// TIA Portal V21 export
FUNCTION "CipEvents" : Void   // FC2, LAD
{ S7_Optimized_Access := 'TRUE' }
// stored: SetENOAutomatically false
   VAR_TEMP   // added for the SCL form of the ladder/FBD networks
      _w1 : Bool;
      _w2 : Bool;
      _w3 : Bool;
      _w4 : Bool;
      _w5 : Bool;
      _w6 : Bool;
      _w7 : Bool;
      _w8 : Bool;
      _w9 : Bool;
      _w10 : Bool;
      _w11 : Bool;
      _w12 : Bool;
      _w13 : Bool;
      _w14 : Bool;
      _w15 : Bool;
      _w16 : Bool;
      _w17 : Bool;
      _w18 : Bool;
      _w19 : Bool;
      _w20 : Bool;
      _w21 : Bool;
      _w22 : Bool;
      _w23 : Bool;
      _w24 : Bool;
      _w25 : Bool;
      _w26 : Bool;
      _w27 : Bool;
      _w28 : Bool;
      _w29 : Bool;
      _w30 : Bool;
      _w31 : Bool;
      _w32 : Bool;
      _w33 : Bool;
      _w34 : Bool;
      _w35 : Bool;
      _w36 : Bool;
      _w37 : Bool;
      _w38 : Bool;
      _w39 : Bool;
      _w40 : Bool;
   END_VAR
BEGIN

REGION Network 1: ****************D500****************
END_REGION

REGION Network 2: Events And Line Print
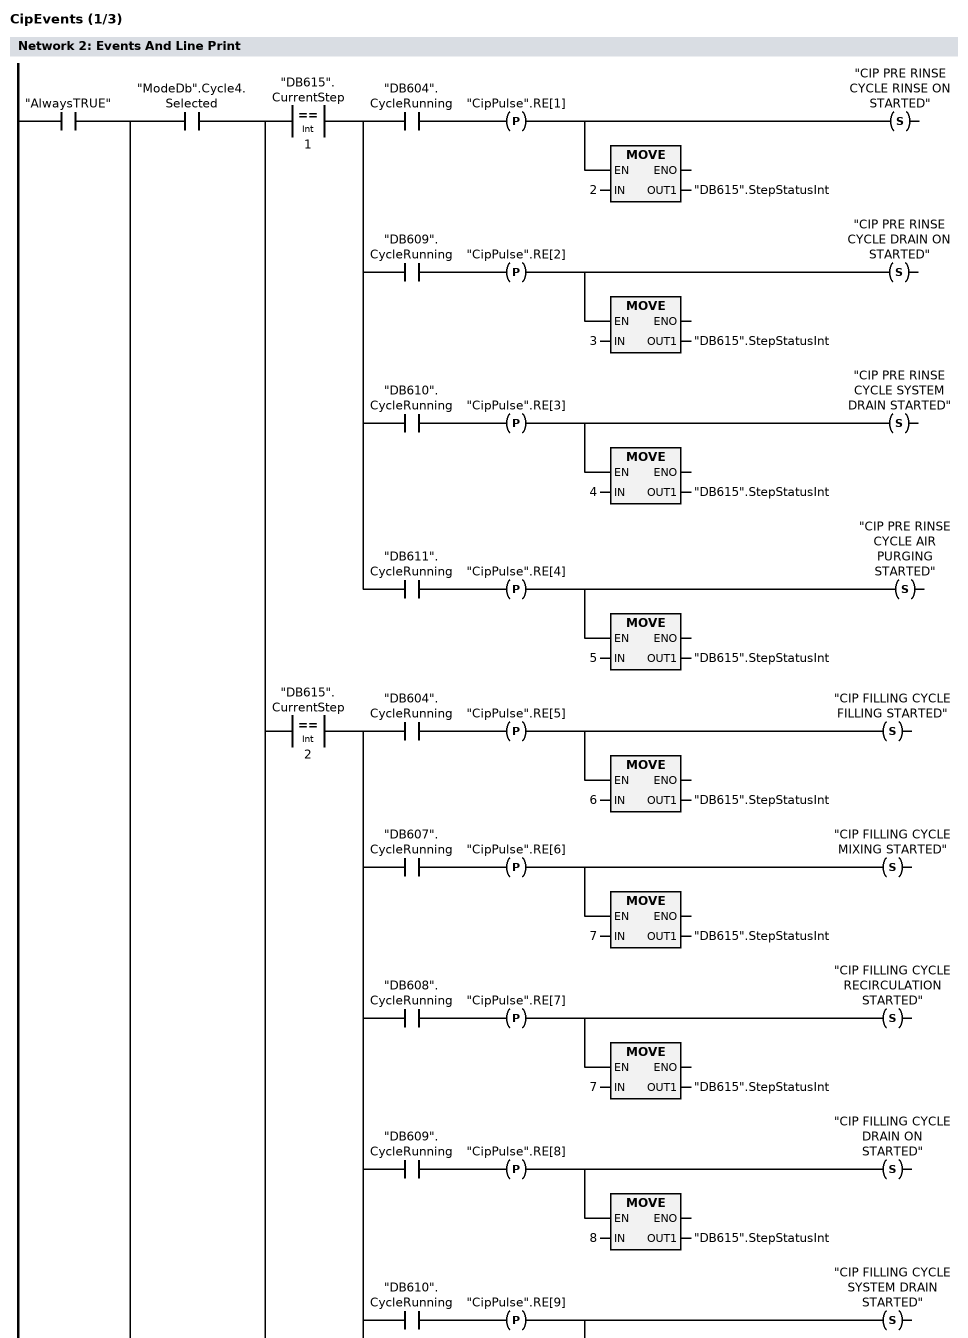
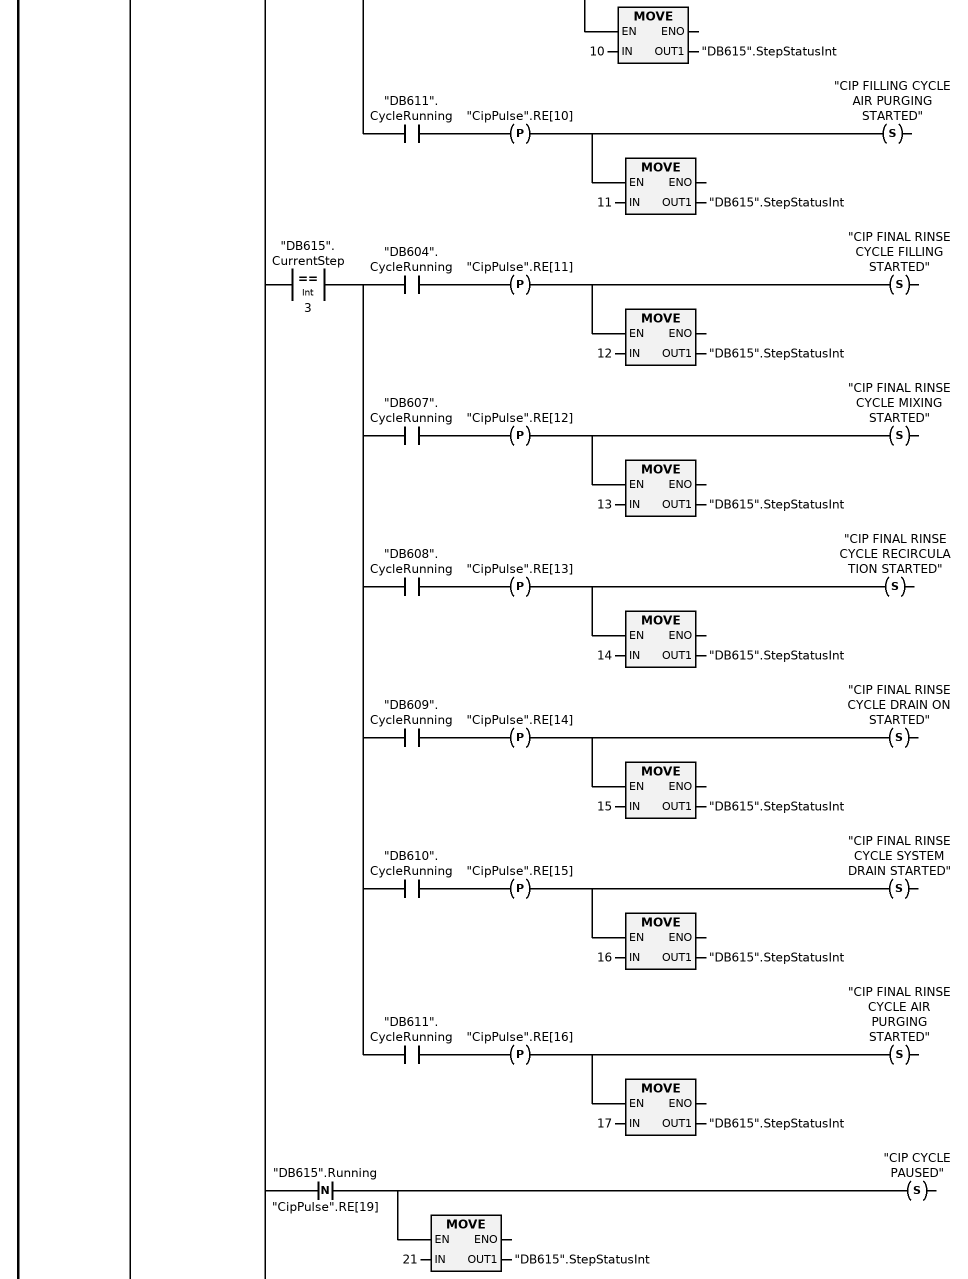
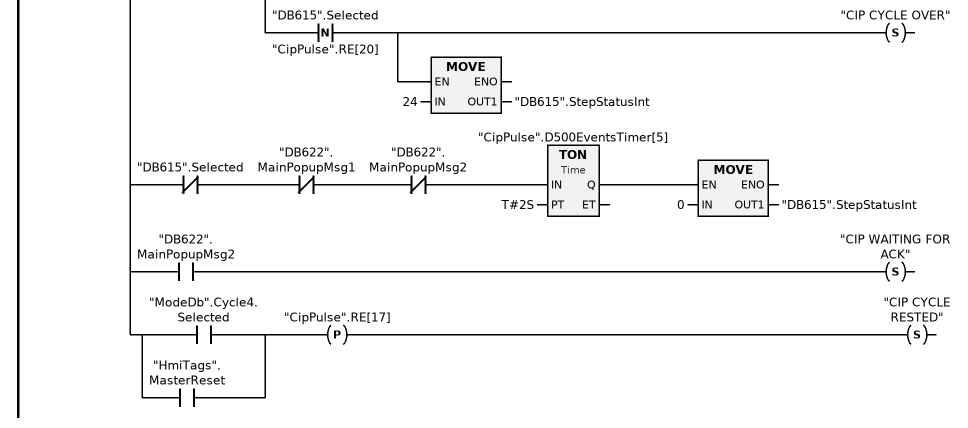
   RUNG wire#powerrail
      Contact( "AlwaysTRUE" )
      wire#w1
      Contact( "ModeDb".Cycle4.Selected )
      wire#w2
      { S7_Templates := "SrcType := Int" } EQ_Contact(in1 := "DB615".CurrentStep, in2 := 1)
      wire#w3
      Contact( "DB604".CycleRunning )
      P_Trig( "CipPulse".RE[1] )
      wire#w4
      S_Coil( "CIP PRE RINSE CYCLE RINSE ON STARTED" )
   END_RUNG
   RUNG wire#w4
      Move(in := 2, out1 => "DB615".StepStatusInt)
   END_RUNG
   RUNG wire#w3
      Contact( "DB609".CycleRunning )
      P_Trig( "CipPulse".RE[2] )
      wire#w5
      S_Coil( "CIP PRE RINSE CYCLE DRAIN ON STARTED" )
   END_RUNG
   RUNG wire#w5
      Move(in := 3, out1 => "DB615".StepStatusInt)
   END_RUNG
   RUNG wire#w3
      Contact( "DB610".CycleRunning )
      P_Trig( "CipPulse".RE[3] )
      wire#w6
      S_Coil( "CIP PRE RINSE CYCLE SYSTEM DRAIN STARTED" )
   END_RUNG
   RUNG wire#w6
      Move(in := 4, out1 => "DB615".StepStatusInt)
   END_RUNG
   RUNG wire#w3
      Contact( "DB611".CycleRunning )
      P_Trig( "CipPulse".RE[4] )
      wire#w7
      S_Coil( "CIP PRE RINSE CYCLE AIR PURGING STARTED" )
   END_RUNG
   RUNG wire#w7
      Move(in := 5, out1 => "DB615".StepStatusInt)
   END_RUNG
   RUNG wire#w2
      { S7_Templates := "SrcType := Int" } EQ_Contact(in1 := "DB615".CurrentStep, in2 := 2)
      wire#w8
      Contact( "DB604".CycleRunning )
      P_Trig( "CipPulse".RE[5] )
      wire#w9
      S_Coil( "CIP FILLING CYCLE FILLING STARTED" )
   END_RUNG
   RUNG wire#w9
      Move(in := 6, out1 => "DB615".StepStatusInt)
   END_RUNG
   RUNG wire#w8
      Contact( "DB607".CycleRunning )
      P_Trig( "CipPulse".RE[6] )
      wire#w10
      S_Coil( "CIP FILLING CYCLE MIXING STARTED" )
   END_RUNG
   RUNG wire#w10
      Move(in := 7, out1 => "DB615".StepStatusInt)
   END_RUNG
   RUNG wire#w8
      Contact( "DB608".CycleRunning )
      P_Trig( "CipPulse".RE[7] )
      wire#w11
      S_Coil( "CIP FILLING CYCLE RECIRCULATION STARTED" )
   END_RUNG
   RUNG wire#w11
      Move(in := 7, out1 => "DB615".StepStatusInt)
   END_RUNG
   RUNG wire#w8
      Contact( "DB609".CycleRunning )
      P_Trig( "CipPulse".RE[8] )
      wire#w12
      S_Coil( "CIP FILLING CYCLE DRAIN ON STARTED" )
   END_RUNG
   RUNG wire#w12
      Move(in := 8, out1 => "DB615".StepStatusInt)
   END_RUNG
   RUNG wire#w8
      Contact( "DB610".CycleRunning )
      P_Trig( "CipPulse".RE[9] )
      wire#w13
      S_Coil( "CIP FILLING CYCLE SYSTEM DRAIN STARTED" )
   END_RUNG
   RUNG wire#w13
      Move(in := 10, out1 => "DB615".StepStatusInt)
   END_RUNG
   RUNG wire#w8
      Contact( "DB611".CycleRunning )
      P_Trig( "CipPulse".RE[10] )
      wire#w14
      S_Coil( "CIP FILLING CYCLE AIR PURGING STARTED" )
   END_RUNG
   RUNG wire#w14
      Move(in := 11, out1 => "DB615".StepStatusInt)
   END_RUNG
   RUNG wire#w2
      { S7_Templates := "SrcType := Int" } EQ_Contact(in1 := "DB615".CurrentStep, in2 := 3)
      wire#w15
      Contact( "DB604".CycleRunning )
      P_Trig( "CipPulse".RE[11] )
      wire#w16
      S_Coil( "CIP FINAL RINSE CYCLE FILLING STARTED" )
   END_RUNG
   RUNG wire#w16
      Move(in := 12, out1 => "DB615".StepStatusInt)
   END_RUNG
   RUNG wire#w15
      Contact( "DB607".CycleRunning )
      P_Trig( "CipPulse".RE[12] )
      wire#w17
      S_Coil( "CIP FINAL RINSE CYCLE MIXING STARTED" )
   END_RUNG
   RUNG wire#w17
      Move(in := 13, out1 => "DB615".StepStatusInt)
   END_RUNG
   RUNG wire#w15
      Contact( "DB608".CycleRunning )
      P_Trig( "CipPulse".RE[13] )
      wire#w18
      S_Coil( "CIP FINAL RINSE CYCLE RECIRCULATION STARTED" )
   END_RUNG
   RUNG wire#w18
      Move(in := 14, out1 => "DB615".StepStatusInt)
   END_RUNG
   RUNG wire#w15
      Contact( "DB609".CycleRunning )
      P_Trig( "CipPulse".RE[14] )
      wire#w19
      S_Coil( "CIP FINAL RINSE CYCLE DRAIN ON STARTED" )
   END_RUNG
   RUNG wire#w19
      Move(in := 15, out1 => "DB615".StepStatusInt)
   END_RUNG
   RUNG wire#w15
      Contact( "DB610".CycleRunning )
      P_Trig( "CipPulse".RE[15] )
      wire#w20
      S_Coil( "CIP FINAL RINSE CYCLE SYSTEM DRAIN STARTED" )
   END_RUNG
   RUNG wire#w20
      Move(in := 16, out1 => "DB615".StepStatusInt)
   END_RUNG
   RUNG wire#w15
      Contact( "DB611".CycleRunning )
      P_Trig( "CipPulse".RE[16] )
      wire#w21
      S_Coil( "CIP FINAL RINSE CYCLE AIR PURGING STARTED" )
   END_RUNG
   RUNG wire#w21
      Move(in := 17, out1 => "DB615".StepStatusInt)
   END_RUNG
   RUNG wire#w2
      N_Contact(operand := "DB615".Running, bit := "CipPulse".RE[19])
      wire#w22
      S_Coil( "CIP CYCLE PAUSED" )
   END_RUNG
   RUNG wire#w22
      Move(in := 21, out1 => "DB615".StepStatusInt)
   END_RUNG
   RUNG wire#w2
      N_Contact(operand := "DB615".Selected, bit := "CipPulse".RE[20])
      wire#w23
      S_Coil( "CIP CYCLE OVER" )
   END_RUNG
   RUNG wire#w23
      Move(in := 24, out1 => "DB615".StepStatusInt)
   END_RUNG
   RUNG wire#w1
      I_Contact( "DB615".Selected )
      I_Contact( "DB622".MainPopupMsg1 )
      I_Contact( "DB622".MainPopupMsg2 )
      { S7_Templates := "time_type := Time" } "CipPulse".D500EventsTimer[5].TON(pt := T#2S, et =>)
      Move(in := 0, out1 => "DB615".StepStatusInt)
   END_RUNG
   RUNG wire#w1
      Contact( "DB622".MainPopupMsg2 )
      S_Coil( "CIP WAITING FOR ACK" )
   END_RUNG
   RUNG wire#w1
      Contact( "ModeDb".Cycle4.Selected )
      wire#w24
      P_Trig( "CipPulse".RE[17] )
      S_Coil( "CIP CYCLE RESTED" )
   END_RUNG
   RUNG wire#w1
      Contact( "HmiTags".MasterReset )
   END_RUNG wire#w24
   // the same network as SCL:
   #_w1 := "AlwaysTRUE" AND "ModeDb".Cycle4.Selected;
   #_w2 := #_w1 AND ("DB615".CurrentStep = 1);
   #_w3 := #_w2 AND "DB604".CycleRunning;
   #_w4 := #_w3 AND NOT "CipPulse".RE[1];   // rising edge
   "CipPulse".RE[1] := #_w3;
   IF #_w4 THEN
       "CIP PRE RINSE CYCLE RINSE ON STARTED" := TRUE;
       "DB615".StepStatusInt := 2;
   END_IF;
   #_w5 := #_w2 AND "DB609".CycleRunning;
   #_w6 := #_w5 AND NOT "CipPulse".RE[2];   // rising edge
   "CipPulse".RE[2] := #_w5;
   IF #_w6 THEN
       "CIP PRE RINSE CYCLE DRAIN ON STARTED" := TRUE;
       "DB615".StepStatusInt := 3;
   END_IF;
   #_w7 := #_w2 AND "DB610".CycleRunning;
   #_w8 := #_w7 AND NOT "CipPulse".RE[3];   // rising edge
   "CipPulse".RE[3] := #_w7;
   IF #_w8 THEN
       "CIP PRE RINSE CYCLE SYSTEM DRAIN STARTED" := TRUE;
       "DB615".StepStatusInt := 4;
   END_IF;
   #_w9 := #_w2 AND "DB611".CycleRunning;
   #_w10 := #_w9 AND NOT "CipPulse".RE[4];   // rising edge
   "CipPulse".RE[4] := #_w9;
   IF #_w10 THEN
       "CIP PRE RINSE CYCLE AIR PURGING STARTED" := TRUE;
       "DB615".StepStatusInt := 5;
   END_IF;
   #_w11 := #_w1 AND ("DB615".CurrentStep = 2);
   #_w12 := #_w11 AND "DB604".CycleRunning;
   #_w13 := #_w12 AND NOT "CipPulse".RE[5];   // rising edge
   "CipPulse".RE[5] := #_w12;
   IF #_w13 THEN
       "CIP FILLING CYCLE FILLING STARTED" := TRUE;
       "DB615".StepStatusInt := 6;
   END_IF;
   #_w14 := #_w11 AND "DB607".CycleRunning;
   #_w15 := #_w14 AND NOT "CipPulse".RE[6];   // rising edge
   "CipPulse".RE[6] := #_w14;
   IF #_w15 THEN
       "CIP FILLING CYCLE MIXING STARTED" := TRUE;
       "DB615".StepStatusInt := 7;
   END_IF;
   #_w16 := #_w11 AND "DB608".CycleRunning;
   #_w17 := #_w16 AND NOT "CipPulse".RE[7];   // rising edge
   "CipPulse".RE[7] := #_w16;
   IF #_w17 THEN
       "CIP FILLING CYCLE RECIRCULATION STARTED" := TRUE;
       "DB615".StepStatusInt := 7;
   END_IF;
   #_w18 := #_w11 AND "DB609".CycleRunning;
   #_w19 := #_w18 AND NOT "CipPulse".RE[8];   // rising edge
   "CipPulse".RE[8] := #_w18;
   IF #_w19 THEN
       "CIP FILLING CYCLE DRAIN ON STARTED" := TRUE;
       "DB615".StepStatusInt := 8;
   END_IF;
   #_w20 := #_w11 AND "DB610".CycleRunning;
   #_w21 := #_w20 AND NOT "CipPulse".RE[9];   // rising edge
   "CipPulse".RE[9] := #_w20;
   IF #_w21 THEN
       "CIP FILLING CYCLE SYSTEM DRAIN STARTED" := TRUE;
       "DB615".StepStatusInt := 10;
   END_IF;
   #_w22 := #_w11 AND "DB611".CycleRunning;
   #_w23 := #_w22 AND NOT "CipPulse".RE[10];   // rising edge
   "CipPulse".RE[10] := #_w22;
   IF #_w23 THEN
       "CIP FILLING CYCLE AIR PURGING STARTED" := TRUE;
       "DB615".StepStatusInt := 11;
   END_IF;
   #_w24 := #_w1 AND ("DB615".CurrentStep = 3);
   #_w25 := #_w24 AND "DB604".CycleRunning;
   #_w26 := #_w25 AND NOT "CipPulse".RE[11];   // rising edge
   "CipPulse".RE[11] := #_w25;
   IF #_w26 THEN
       "CIP FINAL RINSE CYCLE FILLING STARTED" := TRUE;
       "DB615".StepStatusInt := 12;
   END_IF;
   #_w27 := #_w24 AND "DB607".CycleRunning;
   #_w28 := #_w27 AND NOT "CipPulse".RE[12];   // rising edge
   "CipPulse".RE[12] := #_w27;
   IF #_w28 THEN
       "CIP FINAL RINSE CYCLE MIXING STARTED" := TRUE;
       "DB615".StepStatusInt := 13;
   END_IF;
   #_w29 := #_w24 AND "DB608".CycleRunning;
   #_w30 := #_w29 AND NOT "CipPulse".RE[13];   // rising edge
   "CipPulse".RE[13] := #_w29;
   IF #_w30 THEN
       "CIP FINAL RINSE CYCLE RECIRCULATION STARTED" := TRUE;
       "DB615".StepStatusInt := 14;
   END_IF;
   #_w31 := #_w24 AND "DB609".CycleRunning;
   #_w32 := #_w31 AND NOT "CipPulse".RE[14];   // rising edge
   "CipPulse".RE[14] := #_w31;
   IF #_w32 THEN
       "CIP FINAL RINSE CYCLE DRAIN ON STARTED" := TRUE;
       "DB615".StepStatusInt := 15;
   END_IF;
   #_w33 := #_w24 AND "DB610".CycleRunning;
   #_w34 := #_w33 AND NOT "CipPulse".RE[15];   // rising edge
   "CipPulse".RE[15] := #_w33;
   IF #_w34 THEN
       "CIP FINAL RINSE CYCLE SYSTEM DRAIN STARTED" := TRUE;
       "DB615".StepStatusInt := 16;
   END_IF;
   #_w35 := #_w24 AND "DB611".CycleRunning;
   #_w36 := #_w35 AND NOT "CipPulse".RE[16];   // rising edge
   "CipPulse".RE[16] := #_w35;
   IF #_w36 THEN
       "CIP FINAL RINSE CYCLE AIR PURGING STARTED" := TRUE;
       "DB615".StepStatusInt := 17;
   END_IF;
   #_w37 := #_w1 AND NOT "DB615".Running AND "CipPulse".RE[19];   // falling edge of "DB615".Running
   "CipPulse".RE[19] := "DB615".Running;
   IF #_w37 THEN
       "CIP CYCLE PAUSED" := TRUE;
       "DB615".StepStatusInt := 21;
   END_IF;
   #_w38 := #_w1 AND NOT "DB615".Selected AND "CipPulse".RE[20];   // falling edge of "DB615".Selected
   "CipPulse".RE[20] := "DB615".Selected;
   IF #_w38 THEN
       "CIP CYCLE OVER" := TRUE;
       "DB615".StepStatusInt := 24;
   END_IF;
   "CipPulse".D500EventsTimer[5].TON(IN := "AlwaysTRUE" AND NOT "DB615".Selected AND NOT "DB622".MainPopupMsg1 AND NOT "DB622".MainPopupMsg2,
                           PT := T#2S);
   IF "CipPulse".D500EventsTimer[5].Q THEN "DB615".StepStatusInt := 0; END_IF;
   IF "AlwaysTRUE" AND "DB622".MainPopupMsg2 THEN "CIP WAITING FOR ACK" := TRUE; END_IF;
   #_w39 := "AlwaysTRUE" AND ("ModeDb".Cycle4.Selected OR "HmiTags".MasterReset);
   #_w40 := #_w39 AND NOT "CipPulse".RE[17];   // rising edge
   "CipPulse".RE[17] := #_w39;
   IF #_w40 THEN "CIP CYCLE RESTED" := TRUE; END_IF;
END_REGION

REGION Network 3: PRE RINSE
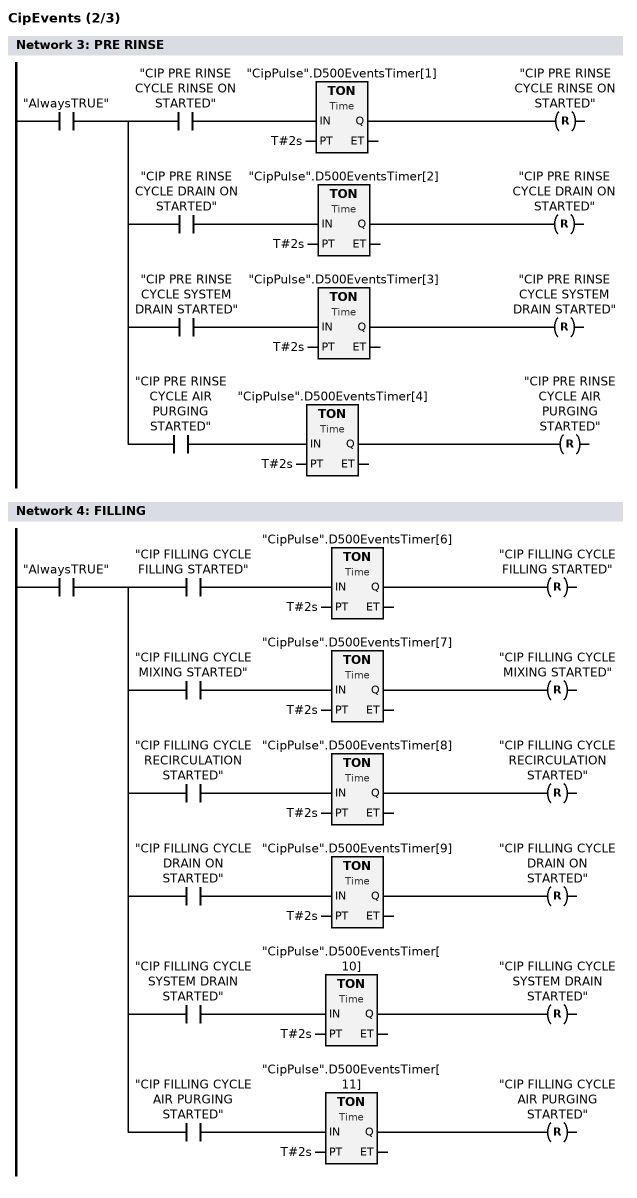
   RUNG wire#powerrail
      Contact( "AlwaysTRUE" )
      wire#w1
      Contact( "CIP PRE RINSE CYCLE RINSE ON STARTED" )
      { S7_Templates := "time_type := Time" } "CipPulse".D500EventsTimer[1].TON(pt := T#2s, et =>)
      R_Coil( "CIP PRE RINSE CYCLE RINSE ON STARTED" )
   END_RUNG
   RUNG wire#w1
      Contact( "CIP PRE RINSE CYCLE DRAIN ON STARTED" )
      { S7_Templates := "time_type := Time" } "CipPulse".D500EventsTimer[2].TON(pt := T#2s, et =>)
      R_Coil( "CIP PRE RINSE CYCLE DRAIN ON STARTED" )
   END_RUNG
   RUNG wire#w1
      Contact( "CIP PRE RINSE CYCLE SYSTEM DRAIN STARTED" )
      { S7_Templates := "time_type := Time" } "CipPulse".D500EventsTimer[3].TON(pt := T#2s, et =>)
      R_Coil( "CIP PRE RINSE CYCLE SYSTEM DRAIN STARTED" )
   END_RUNG
   RUNG wire#w1
      Contact( "CIP PRE RINSE CYCLE AIR PURGING STARTED" )
      { S7_Templates := "time_type := Time" } "CipPulse".D500EventsTimer[4].TON(pt := T#2s, et =>)
      R_Coil( "CIP PRE RINSE CYCLE AIR PURGING STARTED" )
   END_RUNG
   // the same network as SCL:
   "CipPulse".D500EventsTimer[1].TON(IN := "AlwaysTRUE" AND "CIP PRE RINSE CYCLE RINSE ON STARTED", PT := T#2s);
   IF "CipPulse".D500EventsTimer[1].Q THEN "CIP PRE RINSE CYCLE RINSE ON STARTED" := FALSE; END_IF;
   "CipPulse".D500EventsTimer[2].TON(IN := "AlwaysTRUE" AND "CIP PRE RINSE CYCLE DRAIN ON STARTED", PT := T#2s);
   IF "CipPulse".D500EventsTimer[2].Q THEN "CIP PRE RINSE CYCLE DRAIN ON STARTED" := FALSE; END_IF;
   "CipPulse".D500EventsTimer[3].TON(IN := "AlwaysTRUE" AND "CIP PRE RINSE CYCLE SYSTEM DRAIN STARTED",
                           PT := T#2s);
   IF "CipPulse".D500EventsTimer[3].Q THEN "CIP PRE RINSE CYCLE SYSTEM DRAIN STARTED" := FALSE; END_IF;
   "CipPulse".D500EventsTimer[4].TON(IN := "AlwaysTRUE" AND "CIP PRE RINSE CYCLE AIR PURGING STARTED",
                           PT := T#2s);
   IF "CipPulse".D500EventsTimer[4].Q THEN "CIP PRE RINSE CYCLE AIR PURGING STARTED" := FALSE; END_IF;
END_REGION

REGION Network 4: FILLING
   RUNG wire#powerrail
      Contact( "AlwaysTRUE" )
      wire#w1
      Contact( "CIP FILLING CYCLE FILLING STARTED" )
      { S7_Templates := "time_type := Time" } "CipPulse".D500EventsTimer[6].TON(pt := T#2s, et =>)
      R_Coil( "CIP FILLING CYCLE FILLING STARTED" )
   END_RUNG
   RUNG wire#w1
      Contact( "CIP FILLING CYCLE MIXING STARTED" )
      { S7_Templates := "time_type := Time" } "CipPulse".D500EventsTimer[7].TON(pt := T#2s, et =>)
      R_Coil( "CIP FILLING CYCLE MIXING STARTED" )
   END_RUNG
   RUNG wire#w1
      Contact( "CIP FILLING CYCLE RECIRCULATION STARTED" )
      { S7_Templates := "time_type := Time" } "CipPulse".D500EventsTimer[8].TON(pt := T#2s, et =>)
      R_Coil( "CIP FILLING CYCLE RECIRCULATION STARTED" )
   END_RUNG
   RUNG wire#w1
      Contact( "CIP FILLING CYCLE DRAIN ON STARTED" )
      { S7_Templates := "time_type := Time" } "CipPulse".D500EventsTimer[9].TON(pt := T#2s, et =>)
      R_Coil( "CIP FILLING CYCLE DRAIN ON STARTED" )
   END_RUNG
   RUNG wire#w1
      Contact( "CIP FILLING CYCLE SYSTEM DRAIN STARTED" )
      { S7_Templates := "time_type := Time" } "CipPulse".D500EventsTimer[10].TON(pt := T#2s, et =>)
      R_Coil( "CIP FILLING CYCLE SYSTEM DRAIN STARTED" )
   END_RUNG
   RUNG wire#w1
      Contact( "CIP FILLING CYCLE AIR PURGING STARTED" )
      { S7_Templates := "time_type := Time" } "CipPulse".D500EventsTimer[11].TON(pt := T#2s, et =>)
      R_Coil( "CIP FILLING CYCLE AIR PURGING STARTED" )
   END_RUNG
   // the same network as SCL:
   "CipPulse".D500EventsTimer[6].TON(IN := "AlwaysTRUE" AND "CIP FILLING CYCLE FILLING STARTED", PT := T#2s);
   IF "CipPulse".D500EventsTimer[6].Q THEN "CIP FILLING CYCLE FILLING STARTED" := FALSE; END_IF;
   "CipPulse".D500EventsTimer[7].TON(IN := "AlwaysTRUE" AND "CIP FILLING CYCLE MIXING STARTED", PT := T#2s);
   IF "CipPulse".D500EventsTimer[7].Q THEN "CIP FILLING CYCLE MIXING STARTED" := FALSE; END_IF;
   "CipPulse".D500EventsTimer[8].TON(IN := "AlwaysTRUE" AND "CIP FILLING CYCLE RECIRCULATION STARTED",
                           PT := T#2s);
   IF "CipPulse".D500EventsTimer[8].Q THEN "CIP FILLING CYCLE RECIRCULATION STARTED" := FALSE; END_IF;
   "CipPulse".D500EventsTimer[9].TON(IN := "AlwaysTRUE" AND "CIP FILLING CYCLE DRAIN ON STARTED", PT := T#2s);
   IF "CipPulse".D500EventsTimer[9].Q THEN "CIP FILLING CYCLE DRAIN ON STARTED" := FALSE; END_IF;
   "CipPulse".D500EventsTimer[10].TON(IN := "AlwaysTRUE" AND "CIP FILLING CYCLE SYSTEM DRAIN STARTED",
                           PT := T#2s);
   IF "CipPulse".D500EventsTimer[10].Q THEN "CIP FILLING CYCLE SYSTEM DRAIN STARTED" := FALSE; END_IF;
   "CipPulse".D500EventsTimer[11].TON(IN := "AlwaysTRUE" AND "CIP FILLING CYCLE AIR PURGING STARTED",
                           PT := T#2s);
   IF "CipPulse".D500EventsTimer[11].Q THEN "CIP FILLING CYCLE AIR PURGING STARTED" := FALSE; END_IF;
END_REGION

REGION Network 5: FINAL RINSE
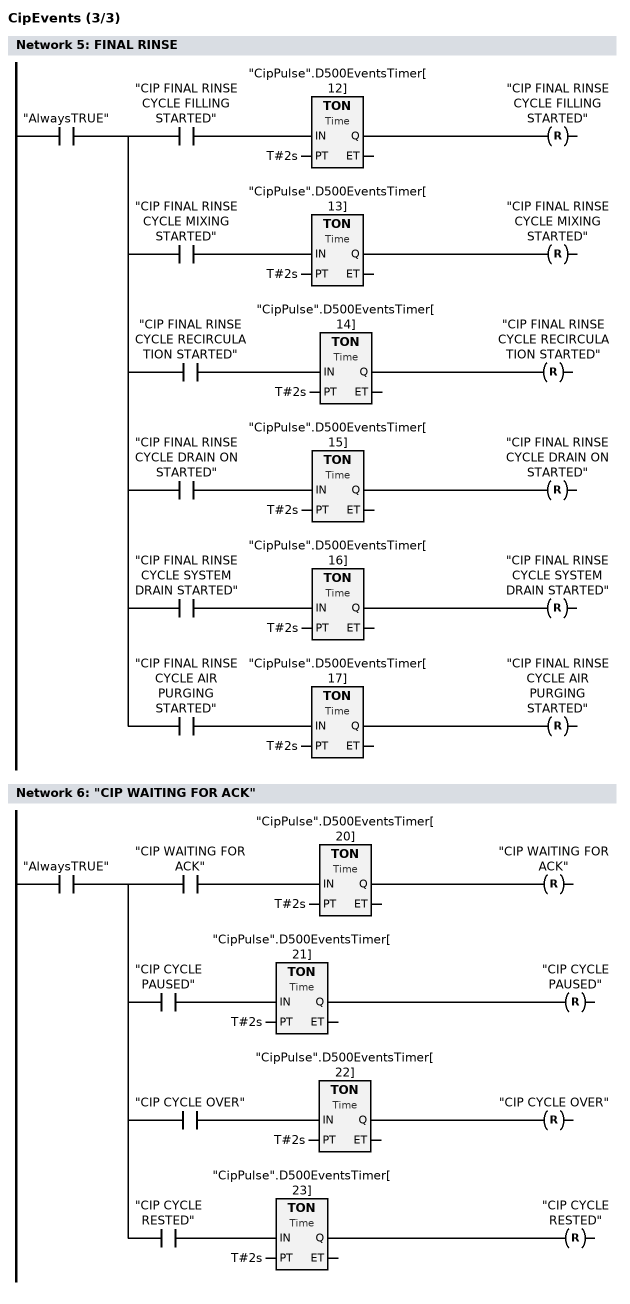
   RUNG wire#powerrail
      Contact( "AlwaysTRUE" )
      wire#w1
      Contact( "CIP FINAL RINSE CYCLE FILLING STARTED" )
      { S7_Templates := "time_type := Time" } "CipPulse".D500EventsTimer[12].TON(pt := T#2s, et =>)
      R_Coil( "CIP FINAL RINSE CYCLE FILLING STARTED" )
   END_RUNG
   RUNG wire#w1
      Contact( "CIP FINAL RINSE CYCLE MIXING STARTED" )
      { S7_Templates := "time_type := Time" } "CipPulse".D500EventsTimer[13].TON(pt := T#2s, et =>)
      R_Coil( "CIP FINAL RINSE CYCLE MIXING STARTED" )
   END_RUNG
   RUNG wire#w1
      Contact( "CIP FINAL RINSE CYCLE RECIRCULATION STARTED" )
      { S7_Templates := "time_type := Time" } "CipPulse".D500EventsTimer[14].TON(pt := T#2s, et =>)
      R_Coil( "CIP FINAL RINSE CYCLE RECIRCULATION STARTED" )
   END_RUNG
   RUNG wire#w1
      Contact( "CIP FINAL RINSE CYCLE DRAIN ON STARTED" )
      { S7_Templates := "time_type := Time" } "CipPulse".D500EventsTimer[15].TON(pt := T#2s, et =>)
      R_Coil( "CIP FINAL RINSE CYCLE DRAIN ON STARTED" )
   END_RUNG
   RUNG wire#w1
      Contact( "CIP FINAL RINSE CYCLE SYSTEM DRAIN STARTED" )
      { S7_Templates := "time_type := Time" } "CipPulse".D500EventsTimer[16].TON(pt := T#2s, et =>)
      R_Coil( "CIP FINAL RINSE CYCLE SYSTEM DRAIN STARTED" )
   END_RUNG
   RUNG wire#w1
      Contact( "CIP FINAL RINSE CYCLE AIR PURGING STARTED" )
      { S7_Templates := "time_type := Time" } "CipPulse".D500EventsTimer[17].TON(pt := T#2s, et =>)
      R_Coil( "CIP FINAL RINSE CYCLE AIR PURGING STARTED" )
   END_RUNG
   // the same network as SCL:
   "CipPulse".D500EventsTimer[12].TON(IN := "AlwaysTRUE" AND "CIP FINAL RINSE CYCLE FILLING STARTED",
                           PT := T#2s);
   IF "CipPulse".D500EventsTimer[12].Q THEN "CIP FINAL RINSE CYCLE FILLING STARTED" := FALSE; END_IF;
   "CipPulse".D500EventsTimer[13].TON(IN := "AlwaysTRUE" AND "CIP FINAL RINSE CYCLE MIXING STARTED", PT := T#2s);
   IF "CipPulse".D500EventsTimer[13].Q THEN "CIP FINAL RINSE CYCLE MIXING STARTED" := FALSE; END_IF;
   "CipPulse".D500EventsTimer[14].TON(IN := "AlwaysTRUE" AND "CIP FINAL RINSE CYCLE RECIRCULATION STARTED",
                           PT := T#2s);
   IF "CipPulse".D500EventsTimer[14].Q THEN "CIP FINAL RINSE CYCLE RECIRCULATION STARTED" := FALSE; END_IF;
   "CipPulse".D500EventsTimer[15].TON(IN := "AlwaysTRUE" AND "CIP FINAL RINSE CYCLE DRAIN ON STARTED",
                           PT := T#2s);
   IF "CipPulse".D500EventsTimer[15].Q THEN "CIP FINAL RINSE CYCLE DRAIN ON STARTED" := FALSE; END_IF;
   "CipPulse".D500EventsTimer[16].TON(IN := "AlwaysTRUE" AND "CIP FINAL RINSE CYCLE SYSTEM DRAIN STARTED",
                           PT := T#2s);
   IF "CipPulse".D500EventsTimer[16].Q THEN "CIP FINAL RINSE CYCLE SYSTEM DRAIN STARTED" := FALSE; END_IF;
   "CipPulse".D500EventsTimer[17].TON(IN := "AlwaysTRUE" AND "CIP FINAL RINSE CYCLE AIR PURGING STARTED",
                           PT := T#2s);
   IF "CipPulse".D500EventsTimer[17].Q THEN "CIP FINAL RINSE CYCLE AIR PURGING STARTED" := FALSE; END_IF;
END_REGION

REGION Network 6: "CIP WAITING FOR ACK"
   RUNG wire#powerrail
      Contact( "AlwaysTRUE" )
      wire#w1
      Contact( "CIP WAITING FOR ACK" )
      { S7_Templates := "time_type := Time" } "CipPulse".D500EventsTimer[20].TON(pt := T#2s, et =>)
      R_Coil( "CIP WAITING FOR ACK" )
   END_RUNG
   RUNG wire#w1
      Contact( "CIP CYCLE PAUSED" )
      { S7_Templates := "time_type := Time" } "CipPulse".D500EventsTimer[21].TON(pt := T#2s, et =>)
      R_Coil( "CIP CYCLE PAUSED" )
   END_RUNG
   RUNG wire#w1
      Contact( "CIP CYCLE OVER" )
      { S7_Templates := "time_type := Time" } "CipPulse".D500EventsTimer[22].TON(pt := T#2s, et =>)
      R_Coil( "CIP CYCLE OVER" )
   END_RUNG
   RUNG wire#w1
      Contact( "CIP CYCLE RESTED" )
      { S7_Templates := "time_type := Time" } "CipPulse".D500EventsTimer[23].TON(pt := T#2s, et =>)
      R_Coil( "CIP CYCLE RESTED" )
   END_RUNG
   // the same network as SCL:
   "CipPulse".D500EventsTimer[20].TON(IN := "AlwaysTRUE" AND "CIP WAITING FOR ACK", PT := T#2s);
   IF "CipPulse".D500EventsTimer[20].Q THEN "CIP WAITING FOR ACK" := FALSE; END_IF;
   "CipPulse".D500EventsTimer[21].TON(IN := "AlwaysTRUE" AND "CIP CYCLE PAUSED", PT := T#2s);
   IF "CipPulse".D500EventsTimer[21].Q THEN "CIP CYCLE PAUSED" := FALSE; END_IF;
   "CipPulse".D500EventsTimer[22].TON(IN := "AlwaysTRUE" AND "CIP CYCLE OVER", PT := T#2s);
   IF "CipPulse".D500EventsTimer[22].Q THEN "CIP CYCLE OVER" := FALSE; END_IF;
   "CipPulse".D500EventsTimer[23].TON(IN := "AlwaysTRUE" AND "CIP CYCLE RESTED", PT := T#2s);
   IF "CipPulse".D500EventsTimer[23].Q THEN "CIP CYCLE RESTED" := FALSE; END_IF;
END_REGION
END_FUNCTION
